// TIA Portal V17 export
// export: Created 2025-03-05T08:01:55.03805Z, ExportSetting WithDefaults, DisplayName Totally Integrated Automation Portal, DisplayVersion V17 Update 8, DisplayName TIA Portal Openness, DisplayVersion V17 Update 8, DisplayName TIA Portal Version Control Interface, DisplayVersion V17, DisplayName SINAMICS Startdrive Advanced, DisplayVersion V17 SP2, DisplayName SINAMICS Startdrive G110M, G120, G120C, G120D, G120P, G115D, DisplayVersion V17 SP2, DisplayName SINAMICS Startdrive G130, G150, S120, S150, SINAMICS MV, S210, DisplayVersion V17 SP2, DisplayName STEP 7 Professional, DisplayVersion V17 Update 8, DisplayName SINUMERIK ONE STEP 7 Toolbox, DisplayVersion V17 Update 12, DisplayName SINUMERIK 840D sl STEP 7 Toolbox, DisplayVersion V17 Update 12, DisplayName STEP 7 Safety, DisplayVersion V17 Update 6, DisplayName WinCC Advanced, DisplayVersion V17 Update 8
TYPE "LBP_typeInternal1"
TITLE = Internal data type for basic program / Tipo de datos interno para el programa básico / Interner Datentyp für Grundprogramm
// Data type only for internal use in the basic program / Tipo de datos solo para uso interno en el programa básico / Datentyp nur für internen Gebrauch im Grundprogramm
// stored: IsFailsafeCompliant false
   STRUCT
      active : Bool;
      mcpAddress : USInt;
      modeDCK : Bool;
      clientPort : UInt;
      connectionId : CONN_OUC;
      mcpClientReference : Word;
      mcpInPointer : Struct
         DbNumber : Word;
         PointerAddress : DWord;
      END_STRUCT;
      mcpOutPointer : Struct
         DbNumber : Word;
         PointerAddress : DWord;
      END_STRUCT;
      mcpDefaultInLength : UInt;
      mcpDefaultOutLength : UInt;
      useIpAddress : Bool;
      ipAddress : Array[1..4] of USInt;
   END_STRUCT;
END_TYPE
